(* PLC project Generated.project, CODESYS CODESYS V3.5 SP19 Patch 1 *)
(* stored: creationDateTime 2026-09-06T13:00:42.443729, modificationDateTime 2026-09-06T13:00:42.443729 *)

(* ======================================================================= 💾 ST_fbWinchSpeedLearning_Table — Table RETAIN apprentissage vitesse ─────────────────────────────────────────────────────────────── 🎯 Rôle : Matrice {axe x sens x charge/vide x palier} de vitesses apprises 📄 Doc metier : DOC/AF/AF_Partie-10_Fonction_Winch_v2.1.md ======================================================================= *)
TYPE ST_fbWinchSpeedLearning_Table : STRUCT
  Cell : ARRAY[1..2, 1..2, 1..2, 1..5] OF ST_fbWinchSpeedLearning_Cell;  (* [axe][sens][charge][palier] axe : 1=M1, 2=M2 sens : 1=montee, 2=descente charge : 1=vide, 2=charge palier : 1..5 *)
END_STRUCT;
END_TYPE

(* ======================================================================= 💾 ST_fbWinchSpeedLearning_Cell — Cellule de vitesse apprise ─────────────────────────────────────────────────────────────── 🎯 Rôle : Cellule unitaire de la table d'apprentissage vitesse par palier 📄 Doc metier : DOC/AF/AF_Partie-10_Fonction_Winch_v2.1.md ======================================================================= *)
TYPE ST_fbWinchSpeedLearning_Cell : STRUCT
  Valid : BOOL;  (* Cellule validee (vitesse apprise exploitable) *)
  SpeedMps : REAL;  (* Vitesse apprise (m/s) *)
  SampleCount : UDINT;  (* Compteur d'echantillons collectes *)
END_STRUCT;
END_TYPE
